INTERFACE I_NodePreExecuteEvent EXTENDS I_Event

METHOD PUBLIC Cancel
VAR_INPUT
END_VAR
END_METHOD

PROPERTY PUBLIC ExecuteCancelled : BOOL
GET
END_GET
END_PROPERTY

PROPERTY PUBLIC Target : I_Node
GET
END_GET
END_PROPERTY

END_INTERFACE

(* stored: Version 1.1.0.1, ProductVersion 3.1.4024.13
   Itf I_NodePreExecuteEvent: Id {a21bbe85-544e-4050-af3c-b5fde68c233c}
   Method Cancel: Id {66742835-59f7-4170-9e0f-e57af0c875e7}
   Property ExecuteCancelled: Id {6be1476e-7d6c-478e-b7a0-a24a4b0f18c4}
   Get Get: Id {409940dd-45b3-461d-97e1-ac15293ff832}
   Property Target: Id {022707f2-eee0-4d3d-80c1-6d3bc504d77e}
   Get Get: Id {f07e414c-cbbe-4556-9251-82547f03880e} *)
